//CHANGING THESE VARIABLES WILL RESULT IN BROKEN LINKS TO THE HMI!
TYPE ST_HMI_Monitor :
STRUCT
	ConditionalFormatting		: ST_HMI_ConditionalFormatting;
	System						: ST_HMI_Monitor_System;
	Powerstack					: ST_HMI_Monitor_Powerstack;
	enclosure					: ST_HMI_Monitor_enclosure;
	firedetection				: ST_HMI_Monitor_Firedetection;
	IPSU						: ST_HMI_Monitor_IPSU;
	OCP							: ST_HMI_Monitor_OCP;
	UPS							: ST_HMI_Monitor_UPS;
	protections					: ST_HMI_Monitor_protections;
	ZPT							: ST_HMI_Monitor_ZPT;
	Switchgear					: ST_HMI_Monitor_switchgear;
	Battery						: ST_HMI_Monitor_Battery;					
	Limits						: ST_HMI_Monitor_limits;
	Connections					: ST_HMI_Monitor_Connections;
	arraydata					: ST_HMI_Monitor_Arraydata;
	cooling						: ST_HMI_Monitor_CoolingSystem;
	AcDcCharger					: ST_HMI_Monitor_AcDcCharger;
	Powercontroller				: ST_PowerControl_Get;
	GenGridController			: ST_GenGridController_get;
	controlfb					: ST_ControlVars;
	PSB							: ST_HMI_Monitor_PSB;	
	DcLink 						: ST_HMI_Monitor_DcLink;
	b_testBool					: BOOL;
END_STRUCT
END_TYPE

(* stored: Version 1.1.0.1, ProductVersion 3.1.4026.18
   DUT ST_HMI_Monitor: Id {06664f7a-1cae-4e79-bc4f-3a4a05ecc5d8} *)
